(* IEC 61131-3 sources: programs/VI-54/VI-54_20171205/VI-54_20171205/Stations/PLC_VI54/VI-54_171014/Class/SdiasManager (part 2) *)

              // additional info which may be needed by the module
              tempCmd.aPara[2] := ud_BusTime_ns$DINT;
              tempCmd.aPara[3] := to_dint(ManagerInfoBlock.ModuleInfos[ActInitAccessIndex].FPGAVersion);

              // check if device ID is ok
              if pModuleInfo^.pThis^.NewInst(pPara:=#tempCmd, pResult:=#_result) = READY then

                // update default accesses if available
                if ManagerInfoBlock.ModuleInfos[ActInitAccessIndex].ReadAccess.usLength then
                  pModuleInfo^.pDefaultAccesses^.ReadAccess.hiOffset := ManagerInfoBlock.ModuleInfos[ActInitAccessIndex].ReadAccess.hiOffset;
                  pModuleInfo^.pDefaultAccesses^.ReadAccess.usLength := ManagerInfoBlock.ModuleInfos[ActInitAccessIndex].ReadAccess.usLength;
                end_if;

                if ManagerInfoBlock.ModuleInfos[ActInitAccessIndex].WriteAccess.usLength then
                  pModuleInfo^.pDefaultAccesses^.WriteAccess.hiOffset := ManagerInfoBlock.ModuleInfos[ActInitAccessIndex].WriteAccess.hiOffset;
                  pModuleInfo^.pDefaultAccesses^.WriteAccess.usLength := ManagerInfoBlock.ModuleInfos[ActInitAccessIndex].WriteAccess.usLength;
                end_if;

                tempCmd.uiCmd := SDIAS_CMD_INIT_ACCESSES;
                RetcodeIPR := pModuleInfo^.pThis^.NewInst(pPara:=#tempCmd, pResult:=#_result);
                if RetcodeIPR = BUSY then
                  // if any module needs more runs => continue here next time
                  b_ModulInitFinished := FALSE;
                  exit;
                elsif RetcodeIPR = ERROR then
                  LogValue("(SdiasManager::CyWork) Failed to add accesses on SDIAS Place 0x{0}", ActInitAccessIndex);
                end_if;
              end_if;
            end_if;
            pModuleInfo += sizeof(t_ModuleObjectInfo);
            ActInitAccessIndex += 1;
          end_while;
        end_if;

        // if we got all accesse => go on
        if b_ModulInitFinished then
          // only if there are entries
          if ManagerInfoBlock.MappingInfo.MappingInfoNo then
            // if the post init is over and the DOs are not created yet => create them in Rt-SSW
            if b_PostInitFinished then
              InitSSW := _StartRtIsoDOCreation;
            else
              CreateAndModifyIsoDOs();

              InitSSW := _CheckInfoBlock;
            end_if;
          else
            LogError("(SdiasManager::CyWork) No Mapping Info in Info Block of SDIAS Manager found! Unable to continue Initialisation!");
            ErrorInitStep := InitSSW;
            InitSSW := _PrepareError;
            ClassState := _ComponentNotExists;
          end_if;
        end_if;

//**********************************************************************************************************************************************************
      _StartRtIsoDOCreation:
        // create and modify the iso DOs in realtime priority
        RtSSW := _CreateAndModifyDOs;
        InitSSW := _Wait4RtIsoDOCreation;

//**********************************************************************************************************************************************************
      _Wait4RtIsoDOCreation:
        // wait for the DOs to be ready
        if RtSSW = _Wait4DOs then
          InitSSW := _CheckInfoBlock;
        end_if;

//**********************************************************************************************************************************************************
      _CheckInfoBlock:

        // only if there are entries
        if ManagerInfoBlock.MappingInfo.MappingInfoNo then
          if ISOWriteDO.pData & ISOReadDO.pData then

            // on VIs the info is copied into the payload. on local SDIAS we get the info directly from the OS
            if ConnectionType = SDIAS_CON_VIA_VARAN_uC then
              pTaskHelp := TaskInfoDO.pData$^t_TaskInfoReadData;
              WriteTaskInfo.pReadData := #pTaskHelp^.WriteTaskInfo;
              ReadTaskInfo.pReadData  := #pTaskHelp^.ReadTaskInfo;
            else
              WriteTaskInfo.pReadData := #WrTaskInfo;
              ReadTaskInfo.pReadData  := #RdTaskInfo;
            end_if;

            // tell the modules their DeviceID, Serialnumber and check if it's the correct object at this place. if so, give them the access pointers
            pModuleInfo := #ModuleObjInfo[0];
            for i := 0 to MaxPlace do

              // if we have an object with this place
              if pModuleInfo^.pThis then
                // and the µC detected a module at this place
                if IsDeviceBitSet(pDeviceBitMap:=#HardwareConfig.DeviceBitmap[0], Place:=i) then

                  if ManagerInfoBlock.ModuleInfos[i].ModuleID = 16#FFFF then
                    pModuleInfo^.pInitState^ := _SPIError;
                  else
                    // get the init state of the LED of this object
                    TempLEDState := pModuleInfo^.pThis^.LEDControl$USINT;

                    // save the state in the local LED Image

                    // get byte position ouf of place (place 0-3 in byte 0, 4-7 in byte 1,...)
                    ByteNr := i$USINT SHR 2;
                    PosInByte := (i$USINT AND 2#11) SHL 1;
                    AppliLEDStates[ByteNr] := (AppliLEDStates[ByteNr] AND NOT(2#11 SHL PosInByte)) OR (TempLEDState SHL PosInByte);

                    // new device info with length parameter to ensure compatibility
                    tempCmd.uiCmd := SDIAS_CMD_DEVICE_INFO2;
                    tempCmd.aPara[0] := sizeof(HDINT); // length of following parameters

                    // hardware version: for 1.10 (printed on the module) we have to transform 16#01 major and 16#0100 minor (drop high nibbles of minor) to 16#00000110
                    tempCmd.aPara[1] := to_dint((ManagerInfoBlock.ModuleInfos[i].HWVersion SHL 8)            OR
                                        ((ManagerInfoBlock.ModuleInfos[i].HWVersionMidLow  SHR 4) AND 16#F0) OR
                                        ((ManagerInfoBlock.ModuleInfos[i].HWVersionMidLow       ) AND 16#0F));

                    // don't check the return code since this command may not be supported
                    pModuleInfo^.pThis^.NewInst(pPara:=#tempCmd, pResult:=#_result);

                    // send the device info to the module
                    tempCmd.uiCmd := SDIAS_CMD_DEVICE_INFO;
                    tempCmd.aPara[0] := to_dint(ManagerInfoBlock.ModuleInfos[i].ModuleID);
                    tempCmd.aPara[1] := (#ManagerInfoBlock.ModuleInfos[i].SerialNo[0])$DINT;

                    // additional info which may be needed by the module
                    tempCmd.aPara[2] := ud_BusTime_ns$DINT;
                    tempCmd.aPara[3] := to_dint(ManagerInfoBlock.ModuleInfos[i].FPGAVersion);

                    // check if device ID is ok
                    if pModuleInfo^.pThis^.NewInst(pPara:=#tempCmd, pResult:=#_result) = READY then

                      // the module id matches, now check the accesses

                      // update default accesses if available
                      if ManagerInfoBlock.ModuleInfos[i].ReadAccess.usLength then
                        pModuleInfo^.pDefaultAccesses^.ReadAccess.hiOffset := ManagerInfoBlock.ModuleInfos[i].ReadAccess.hiOffset;
                        pModuleInfo^.pDefaultAccesses^.ReadAccess.usLength := ManagerInfoBlock.ModuleInfos[i].ReadAccess.usLength;

                        // store the pointers to the correct payload data for later usage in the SDIAS Client class
                        pModuleInfo^.pDefaultAccesses^.ReadAccess.pControlByte$^void  := ISOWriteDO.pData + ManagerInfoBlock.ModuleInfos[i].ReadDODataWrOffset - ISOWriteDO.Offset;
                        pModuleInfo^.pDefaultAccesses^.ReadAccess.pStateByte$^void    := ISOReadDO.pData  + ManagerInfoBlock.ModuleInfos[i].ReadDODataRdOffset - ISOReadDO.Offset;
                        pModuleInfo^.pDefaultAccesses^.ReadAccess.pData               := ISOReadDO.pData  + ManagerInfoBlock.ModuleInfos[i].ReadDODataRdOffset - ISOReadDO.Offset + sizeof(t_SDIAS_StateByte);
                      end_if;

                      if ManagerInfoBlock.ModuleInfos[i].WriteAccess.usLength then
                        pModuleInfo^.pDefaultAccesses^.WriteAccess.hiOffset := ManagerInfoBlock.ModuleInfos[i].WriteAccess.hiOffset;
                        pModuleInfo^.pDefaultAccesses^.WriteAccess.usLength := ManagerInfoBlock.ModuleInfos[i].WriteAccess.usLength;

                        // store the pointers to the correct payload data for later usage in the SDIAS Client class
                        pModuleInfo^.pDefaultAccesses^.WriteAccess.pControlByte$^void  := ISOWriteDO.pData + ManagerInfoBlock.ModuleInfos[i].WriteDODataWrOffset - ISOWriteDO.Offset;
                        pModuleInfo^.pDefaultAccesses^.WriteAccess.pStateByte$^void    := ISOReadDO.pData + ManagerInfoBlock.ModuleInfos[i].WriteDODataRdOffset - ISOReadDO.Offset;
                        pModuleInfo^.pDefaultAccesses^.WriteAccess.pData               := ISOWriteDO.pData + ManagerInfoBlock.ModuleInfos[i].WriteDODataWrOffset - ISOWriteDO.Offset + sizeof(t_SDIAS_ControlByte);
                      end_if;
                    else
                      // wrong device ID
                      if pModuleInfo^.Required then
                        // first stop blocking the init, otherwise the init freezes when we have a required error
                        if b_PostInitFinished = FALSE then
                          SendPostInitFinished(DisableThisObject:=TRUE);
                        end_if;

                        LogValue("(SdiasManager::CyWork) Wrong device ID at SDIAS Place 0x{0}", i);

                        SetRequiredError(pTargetThis:=pModuleInfo^.pThis, Place:=i);
                      else
                        pModuleInfo^.pInitState^ := _WrongHardware;
                      end_if;
                    end_if;
                  end_if;
                else
                  // module is not in the device bitmap, but we got an object
                  if pModuleInfo^.Required then
                    // first stop blocking the init, otherwise the init freezes when we have a required error
                    if b_PostInitFinished = FALSE then
                      SendPostInitFinished(DisableThisObject:=TRUE);
                    end_if;

                    SetRequiredError(pTargetThis:=pModuleInfo^.pThis, Place:=i);
                  else
                    pModuleInfo^.pInitState^ := _NoHardware;
                  end_if;
                end_if;
              end_if;

              pModuleInfo += sizeof(t_ModuleObjectInfo);
            end_for;
          end_if;

          if ConnectionType = SDIAS_CON_VIA_VARAN_uC then
            InitSSW := _PrepareResetIsoRdPayload;
          else
            // we don't have to reset the payload => done by OS
            udCurCheckedMod := 0;
            InitSSW := _CheckModule_Valid;
          end_if;

        else
          LogError("(SdiasManager::CyWork) No Mapping Info in Info Block of SDIAS Manager found! Unable to continue Initialisation!");
          ErrorInitStep := InitSSW;
          InitSSW := _PrepareError;
          ClassState := _ComponentNotExists;
        end_if;

//**********************************************************************************************************************************************************
      _PrepareResetIsoRdPayload:
        // prepare resetting the read payload (toggle bits)
        AccessProgress := 0;
        // reset the write buffer
        _memset(dest:=ASYWriteDO.pData, usByte:=0, cntr:=128);
        NewDataSize := ISOReadDO.Length;
        if NewDataSize > 128 then
          NewDataSize := 128;
        end_if;

        if ChangeAsyWr(Offset:=ISOReadDO.Offset,
                       Length:=NewDataSize$USINT,
                       RunState:=_BUS_IF_RUN_STATE_CONT_RUN,
                       UsageType:=_UsedBySSW) then

          InitSSW := _ResetIsoRdPayload;
        end_if;

//**********************************************************************************************************************************************************
      _ResetIsoRdPayload:
        AccessProgress += NewDataSize;

        if AccessProgress < ISOReadDO.Length then
          if (ISOReadDO.Length - AccessProgress) > 128 then
            // we need more than 128 bytes => write the next 128
            TempNewDataSize := 128;
          else
            // we need to write the rest (last package)
            TempNewDataSize := (ISOReadDO.Length - AccessProgress);
          end_if;

          if ChangeAsyWr(Offset:=ISOReadDO.Offset + AccessProgress,
                         Length:=TempNewDataSize$USINT,
                         RunState:=_BUS_IF_RUN_STATE_CONT_RUN,
                         UsageType:=_UsedBySSW) then
              NewDataSize := TempNewDataSize;
          else
            NewDataSize := 0;
          end_if;
        else
          // we got the complete info block now => stop the DO
          if ChangeAsyWr(Offset:=0,
                         Length:=0,
                         RunState:=_BUS_IF_RUN_STATE_NO_RUN,
                         UsageType:=_UsedBySSW) then

            InitSSW := _PrepareResetIsoWrPayload;
          else
            NewDataSize := 0;
          end_if;
        end_if;

//**********************************************************************************************************************************************************
      _PrepareResetIsoWrPayload:
        // prepare resetting the read payload (toggle bits)
        AccessProgress := 0;
        // reset the write buffer
        _memset(dest:=ASYWriteDO.pData, usByte:=0, cntr:=128);
        NewDataSize := ISOWriteDO.Length;
        if NewDataSize > 128 then
          NewDataSize := 128;
        end_if;

        if ChangeAsyWr(Offset:=ISOWriteDO.Offset,
                       Length:=NewDataSize$USINT,
                       RunState:=_BUS_IF_RUN_STATE_CONT_RUN,
                       UsageType:=_UsedBySSW) then

          InitSSW := _ResetIsoWrPayload;
        end_if;

//**********************************************************************************************************************************************************
      _ResetIsoWrPayload:
        AccessProgress += NewDataSize;

        if AccessProgress < ISOWriteDO.Length then
          if (ISOWriteDO.Length - AccessProgress) > 128 then
            // we need more than 128 bytes => write the next 128
            TempNewDataSize := 128;
          else
            // we need to write the rest (last package)
            TempNewDataSize := (ISOWriteDO.Length - AccessProgress);
          end_if;

          if ChangeAsyWr(Offset:=ISOWriteDO.Offset + AccessProgress,
                         Length:=TempNewDataSize$USINT,
                         RunState:=_BUS_IF_RUN_STATE_CONT_RUN,
                         UsageType:=_UsedBySSW) then
              NewDataSize := TempNewDataSize;
          else
            NewDataSize := 0;
          end_if;
        else
          // we got the complete info block now => stop the DO
          if ChangeAsyWr(Offset:=0,
                         Length:=0,
                         RunState:=_BUS_IF_RUN_STATE_NO_RUN,
                         UsageType:=_UsedBySSW) then

            udCurCheckedMod := 0;
            InitSSW := _CheckModule_Valid;
          else
            NewDataSize := 0;
          end_if;
        end_if;

//**********************************************************************************************************************************************************
      _CheckModule_Valid:
        // tell the modules their DeviceID, Serialnumber and check if it's the correct object at this place. if so, give them the access pointers
        pModuleInfo := #ModuleObjInfo[udCurCheckedMod];

        // if we have an object with this place
        if pModuleInfo^.pThis then
          // and the µC detected a module at this place
          if IsDeviceBitSet(pDeviceBitMap:=#HardwareConfig.DeviceBitmap[0], Place:=udCurCheckedMod) then

            if ManagerInfoBlock.ModuleInfos[udCurCheckedMod].ModuleID = 16#FFFF then
              // SPI Error
              if pModuleInfo^.Required then
                // first stop blocking the init, otherwise the init freezes when we have a required error
                if b_PostInitFinished = FALSE then
                  SendPostInitFinished(DisableThisObject:=TRUE);
                end_if;

                LogValue("(SdiasManager::CyWork) Wrong device ID at SDIAS Place 0x{0}", udCurCheckedMod);

                SetRequiredError(pTargetThis:=pModuleInfo^.pThis, Place:=udCurCheckedMod);
              else
                pModuleInfo^.pInitState^ := _SPIError;
                InitSSW := _CheckNextModule;
              end_if;
            else
              // get the init state of the LED of this object
              TempLEDState := pModuleInfo^.pThis^.LEDControl$USINT;

              // save the state in the local LED Image

              // get byte position ouf of place (place 0-3 in byte 0, 4-7 in byte 1,...)
              ByteNr := udCurCheckedMod$USINT SHR 2;
              PosInByte := (udCurCheckedMod$USINT AND 2#11) SHL 1;
              AppliLEDStates[ByteNr] := (AppliLEDStates[ByteNr] AND NOT(2#11 SHL PosInByte)) OR (TempLEDState SHL PosInByte);

              // new device info with length parameter to ensure compatibility
              tempCmd.uiCmd := SDIAS_CMD_DEVICE_INFO2;
              tempCmd.aPara[0] := sizeof(HDINT); // length of following parameters

              // hardware version: for 1.10 (printed on the module) we have to transform 16#01 major and 16#0100 minor (drop high nibbles of minor) to 16#00000110
              tempCmd.aPara[1] := to_dint((ManagerInfoBlock.ModuleInfos[udCurCheckedMod].HWVersion SHL 8)            OR
                                  ((ManagerInfoBlock.ModuleInfos[udCurCheckedMod].HWVersionMidLow  SHR 4) AND 16#F0) OR
                                  ((ManagerInfoBlock.ModuleInfos[udCurCheckedMod].HWVersionMidLow       ) AND 16#0F));

              // don't check the return code since this command may not be supported
              pModuleInfo^.pThis^.NewInst(pPara:=#tempCmd, pResult:=#_result);

              // send the device info to the module
              tempCmd.uiCmd := SDIAS_CMD_DEVICE_INFO;
              tempCmd.aPara[0] := to_dint(ManagerInfoBlock.ModuleInfos[udCurCheckedMod].ModuleID);
              tempCmd.aPara[1] := (#ManagerInfoBlock.ModuleInfos[udCurCheckedMod].SerialNo[0])$DINT;

              // additional info which may be needed by the module
              tempCmd.aPara[2] := ud_BusTime_ns$DINT;
              tempCmd.aPara[3] := to_dint(ManagerInfoBlock.ModuleInfos[udCurCheckedMod].FPGAVersion);

              // check if device ID is ok
              if pModuleInfo^.pThis^.NewInst(pPara:=#tempCmd, pResult:=#_result) = READY then

                // the module id matches, continue with access
                pCurCheckModAccPtr := pModuleInfo^.pFirstAccess;
                InitSSW := _SetModAccess;

              else
                // wrong device ID
                if pModuleInfo^.Required then
                  // first stop blocking the init, otherwise the init freezes when we have a required error
                  if b_PostInitFinished = FALSE then
                    SendPostInitFinished(DisableThisObject:=TRUE);
                  end_if;

                  LogValue("(SdiasManager::CyWork) Wrong device ID at SDIAS Place 0x{0}", udCurCheckedMod);

                  SetRequiredError(pTargetThis:=pModuleInfo^.pThis, Place:=udCurCheckedMod);
                else
                  pModuleInfo^.pInitState^ := _WrongHardware;
                  InitSSW := _CheckNextModule;
                end_if;
              end_if;
            end_if;
          else
            // module is not in the device bitmap, but we got an object
            if pModuleInfo^.Required then
              // first stop blocking the init, otherwise the init freezes when we have a required error
              if b_PostInitFinished = FALSE then
                SendPostInitFinished(DisableThisObject:=TRUE);
              end_if;

              SetRequiredError(pTargetThis:=pModuleInfo^.pThis, Place:=udCurCheckedMod);
            else
              pModuleInfo^.pInitState^ := _NoHardware;
              InitSSW := _CheckNextModule;
            end_if;
          end_if;
        else
          InitSSW := _CheckNextModule;
        end_if;

//**********************************************************************************************************************************************************
      _SetModAccess:
        pModuleInfo := #ModuleObjInfo[udCurCheckedMod];
        if pCurCheckModAccPtr = NIL then
          // no special accesses => call connect event and proceed with next module
          pModuleInfo^.pThis^.ConnectEvent();
          InitSSW := _CheckNextModule;
        elsif (pCurCheckModAccPtr^.eAccessType = _Read) | (pCurCheckModAccPtr^.eAccessType = _ReadDynamic) then

          pWaitAccess := pCurCheckModAccPtr^.pWaitForAccess;
          if pWaitAccess <> NIL then
            if (pWaitAccess^.eAccessType <> pCurCheckModAccPtr^.eAccessType) then
              pWaitAccess := NIL;
            end_if;
          end_if;

          if(pWaitAccess <> NIL) then
            // address of state byte
            iWaitOffset := ISOReadDO.Offset + (pWaitAccess^.ppStateByte^$HDINT - ISOReadDO.pData$HDINT)$UINT; //pWaitAccess^.hiDOOffsetInDPRAM;
          else
            iWaitOffset := SDIAS_INVALID_VOLATILE_WAIT_HANDLE;
          end_if;

          // Create access by new funtion
          iRetCode := DOL_Handling_Add_DO_TO_List(bIsWriteAcc0:= 0,
                                                  iModAddr0:= pCurCheckModAccPtr^.hiOffset + (udCurCheckedMod shl 10),
                                                  iDataLen0:= pCurCheckModAccPtr^.uiLength,
                                                  bCtrlAcc0:= pCurCheckModAccPtr^.bCtrlAcc0,
                                                  iWaitDOOffset0:= iWaitOffset,
                                                  bIsDynamic0 := (pCurCheckModAccPtr^.eAccessType = _ReadDynamic),
                                                  pActAccess0 := pCurCheckModAccPtr);

          if iRetCode = 0 then

            // store the pointers to the correct payload data for later usage in the SDIAS Client class
            if pCurCheckModAccPtr^.ppControlByte then
              pCurCheckModAccPtr^.ppControlByte^$^void := ISOWriteDO.pData + gcWrite_DOL_Desc.iOffFirstData + gcMapping_Informations[IsoWrPayload].StartAddress - ISOWriteDO.Offset;
              if pCurCheckModAccPtr^.eAccessType = _ReadDynamic then
                pControlStruct := pCurCheckModAccPtr^.ppControlByte^$^t_SDIAS_ControlStructDynamic;
                pControlStruct^.ControlByte.EnableFlexRead := TRUE;
                pControlStruct^.hiOffset := pCurCheckModAccPtr^.hiOffset + (udCurCheckedMod shl 10);
                pControlStruct^.usLength := pCurCheckModAccPtr^.uiLength$USINT;
              end_if;
            end_if;
            if pCurCheckModAccPtr^.ppStateByte then
              pCurCheckModAccPtr^.ppStateByte^$^void := ISOReadDO.pData + gcRead_DOL_Desc.iOffFirstData + gcMapping_Informations[IsoRdPayload].StartAddress - ISOReadDO.Offset;
            end_if;
            if pCurCheckModAccPtr^.ppData then
              pCurCheckModAccPtr^.ppData^$^void := ISOReadDO.pData + gcRead_DOL_Desc.iOffFirstData + sizeof(t_SDIAS_StateByte) + gcMapping_Informations[IsoRdPayload].StartAddress - ISOReadDO.Offset;;
            end_if;

            InitSSW := _WriteModAccess;
          else
            ErrorInitStep := InitSSW;
            InitSSW := _PrepareError;
            ClassState := _DOCmdInvalid;
          end_if;

        elsif (pCurCheckModAccPtr^.eAccessType = _Write) | (pCurCheckModAccPtr^.eAccessType = _WriteDynamic) then

          pWaitAccess := pCurCheckModAccPtr^.pWaitForAccess;
          if pWaitAccess <> NIL then
            if (pWaitAccess^.eAccessType <> pCurCheckModAccPtr^.eAccessType) then
              pWaitAccess := NIL;
            end_if;
          end_if;

          if(pWaitAccess <> NIL) then
            // address of state byte
            iWaitOffset := ISOReadDO.Offset + (pWaitAccess^.ppStateByte^$HDINT - ISOReadDO.pData$HDINT)$UINT; //pWaitAccess^.hiDOOffsetInDPRAM;
          else
            iWaitOffset := SDIAS_INVALID_VOLATILE_WAIT_HANDLE;
          end_if;

          // Create access by new funtion
          iRetCode := DOL_Handling_Add_DO_TO_List(bIsWriteAcc0:= 1,
                                                  iModAddr0:= pCurCheckModAccPtr^.hiOffset + (udCurCheckedMod shl 10),
                                                  iDataLen0:= pCurCheckModAccPtr^.uiLength,
                                                  bCtrlAcc0:= pCurCheckModAccPtr^.bCtrlAcc0,
                                                  iWaitDOOffset0:= iWaitOffset,
                                                  bIsDynamic0 := (pCurCheckModAccPtr^.eAccessType = _WriteDynamic),
                                                  pActAccess0 := pCurCheckModAccPtr);

          if iRetCode = 0 then
            // store the pointers to the correct payload data for later usage in the SDIAS Client class
            if pCurCheckModAccPtr^.ppControlByte then
              pCurCheckModAccPtr^.ppControlByte^$^void := ISOWriteDO.pData + gcWrite_DOL_Desc.iOffFirstData + gcMapping_Informations[IsoWrPayload].StartAddress - ISOWriteDO.Offset;
              if pCurCheckModAccPtr^.eAccessType = _WriteDynamic then
                pControlStruct := pCurCheckModAccPtr^.ppControlByte^$^t_SDIAS_ControlStructDynamic;
                pControlStruct^.ControlByte.EnableFlexWrite := TRUE;
                pControlStruct^.hiOffset := pCurCheckModAccPtr^.hiOffset + (udCurCheckedMod shl 10);
                pControlStruct^.usLength := pCurCheckModAccPtr^.uiLength$USINT;
              end_if;
            end_if;
            if pCurCheckModAccPtr^.ppStateByte then
              pCurCheckModAccPtr^.ppStateByte^$^void := ISOReadDO.pData + gcRead_DOL_Desc.iOffFirstData + gcMapping_Informations[IsoRdPayload].StartAddress - ISOReadDO.Offset;
            end_if;
            if pCurCheckModAccPtr^.ppData then
              // the data start after the header. at dynamic objects we have more header in write payload => data start after the structure
              if pCurCheckModAccPtr^.eAccessType = _WriteDynamic then
                pCurCheckModAccPtr^.ppData^$^void := ISOWriteDO.pData + gcWrite_DOL_Desc.iOffFirstData + sizeof(t_SDIAS_ControlStructDynamic) + gcMapping_Informations[IsoWrPayload].StartAddress - ISOWriteDO.Offset;
              else
                pCurCheckModAccPtr^.ppData^$^void := ISOWriteDO.pData + gcWrite_DOL_Desc.iOffFirstData + sizeof(t_SDIAS_ControlByte) + gcMapping_Informations[IsoWrPayload].StartAddress - ISOWriteDO.Offset;
              end_if;
            end_if;

            InitSSW := _WriteModAccess;
          else
            ErrorInitStep := InitSSW;
            InitSSW := _PrepareError;
            ClassState := _DOCmdInvalid;
          end_if;
        end_if;

//**********************************************************************************************************************************************************
      _WriteModAccess:

          if ConnectionType = SDIAS_CON_VIA_VARAN_uC then
            ASYWriteDO.pData^$t_SDIAS_DOListEntryX2 := cModulAccessCmds;

            // Write data to manager dpram
            if ChangeAsyWr(Offset   := uiWriteCmdAddr,
                           Length   := sizeof(cModulAccessCmds),
                           RunState := _BUS_IF_RUN_STATE_SINGLE_RUN,
                           UsageType:= _UsedBySSW) then

              InitSSW := _SetNextModAccess;
            end_if;
          else
            // OS already did this for us
            InitSSW := _SetNextModAccess;
          end_if;

//**********************************************************************************************************************************************************
      _SetNextModAccess:

        AsyWriteUsage  := _NotUsed;

        pModuleInfo := #ModuleObjInfo[udCurCheckedMod];
        // Reached last access - trigger connect event
        if(pCurCheckModAccPtr^.pNext = NIL) then
          // call the connect event now (pointers are set now to enable the accesses)
          pModuleInfo^.pThis^.ConnectEvent();
          InitSSW := _CheckNextModule;
        else
          pCurCheckModAccPtr := pCurCheckModAccPtr^.pNext;
          InitSSW := _SetModAccess;
        end_if;

//**********************************************************************************************************************************************************
      _CheckNextModule:

        // Switch to next module
        udCurCheckedMod += 1;

        if(udCurCheckedMod <= MaxPlace) then
          InitSSW := _CheckModule_Valid;
        else
          if ConnectionType = SDIAS_CON_VIA_VARAN_uC then
            InitSSW := _WriteDOL_Offsets;
          else
            // we don't have to reset the payload => done by OS
            if MaxPlace <> SDIAS_PLACE_NO_MODULE_ADDED_SO_FAR then
              InitSSW := _SetStartConfigIsoRd;
            else
              LogError("(SdiasManager::CyWork) No SDIAS Client objects projected/connected to the SDIAS Manager! Unable to continue with Initialisation!");
              ErrorInitStep := InitSSW;
              InitSSW := _PrepareError;
              ClassState := _NoHardware;
            end_if;
          end_if;
        end_if;

//**********************************************************************************************************************************************************
      _WriteDOL_Offsets:

        // Create list informations
        // Read list offsets
        iDataOffsets[0] := gcRead_DOL_Desc.iOffEndCmd;
        iDataOffsets[1] := gcRead_DOL_Desc.iOffLastData;

        // Write list offsets
        iDataOffsets[2] := gcWrite_DOL_Desc.iOffEndCmd;
        iDataOffsets[3] := gcWrite_DOL_Desc.iOffLastData;

        bReceivedNewEndRsp := FALSE;
#ifdef HWK_SHOW_PRAGMA_MESSAGES
#pragma message("RamAnd 23.11.2013 19:17 \ ein neues Ende muss nur geschrieben werden, wenn Spezialzugriffe angelegt wurden")
#endif
        if(AddSDOReq(pCmdSvr:= (#ClassState.pMeth)$^SvrChCmd,
                     Command:= SDIAS_SDO_CMD_SET_NEW_END,
                     Place:= SDIAS_MANAGER_PLACE,
                     CmdLength:= 4* sizeof(UDINT),
                     pReqBuf:= #iDataOffsets[0]$USINT) = READY$DINT) then

           InitSSW := _WaitReq_DOL_Offsets;
        end_if;

//**********************************************************************************************************************************************************
      _WaitReq_DOL_Offsets:
        // Wait until receiving request
        if bReceivedNewEndRsp = TRUE then
          bReceivedNewEndRsp := FALSE;

          InitSSW := _GetEventIDs;
        end_if;

//**********************************************************************************************************************************************************
      _GetEventIDs:
        if MaxPlace <> SDIAS_PLACE_NO_MODULE_ADDED_SO_FAR then
            // we also start a read access here, so we got the data in the next step
          if ChangeAsyRd(Offset:=SDIAS_OFFSET_TASK_EVENT_IDS,
                         Length:=sizeof(t_TaskEventIDs),
                         RunState:=_BUS_IF_RUN_STATE_SINGLE_RUN,
                         UsageType:=_UsedBySSW) then

            udCurCheckedMod := 0;
            InitSSW := _SetStartConfigIsoRd;
          end_if;
        else
          LogError("(SdiasManager::CyWork) No SDIAS Client objects projected/connected to the SDIAS Manager! Unable to continue with Initialisation!");
          ErrorInitStep := InitSSW;
          InitSSW := _PrepareError;
          ClassState := _NoHardware;
        end_if;

//**********************************************************************************************************************************************************
      _SetStartConfigIsoRd:
        if ConnectionType = SDIAS_CON_VIA_VARAN_uC then
          TaskEventIDs := ASYReadDO.pData^$t_TaskEventIDs;
        else
          for i := 0 to 7 do
            if SDIAS_iGetNodePropertyIndex(hNodeHandle    := udNodeHandle
                                    , udIndex             := i
                                    , udPropertyId        := SDM_PROP_TASK_START_EVENT_ID,
                                    , pudPropertyValue    := (#TaskEventIDs[i])$^UDINT
                                    ) <> SDIAS_OK then
              LogValue("(SdiasManager::CyWork) Failed to get task event ID 0x{0} via OS interface!", i);
              ErrorInitStep := InitSSW;
              InitSSW := _PrepareError;
              ClassState := _ManagerError;
              return;
            end_if;
          end_for;
        end_if;

        AsyReadUsage  := _NotUsed;

        // search for the sync out 0 event id
        b_FoundIt := FALSE;
        for i := 0 to 7 do
          if ConnectionType = SDIAS_CON_VIA_VARAN_uC then
            if TaskEventIDs[i] = SDIAS_EVENT_MASK_ID_SYNC_OUT0 then
              b_FoundIt := TRUE;
              exit;
            end_if;
          else
            if TaskEventIDs[i] = SDIAS_EVENT_MASK_ID_SYNC_OUT2 then
              b_FoundIt := TRUE;
              exit;
            end_if;
          end_if;
        end_for;

        // if we found it, use it for the task start config 0 (which is used by the iso read task)
        if b_FoundIt then
          TaskStartConfig.EventSelection := 1 SHL i$USINT;

          // iso read starts 0µs after the sync
          TaskStartConfig.StartDelay_us  := 0;

          if ConnectionType = SDIAS_CON_VIA_VARAN_uC then
            ASYWriteDO.pData^$t_TaskStartConfig := TaskStartConfig;
            if ChangeAsyWr(Offset:=SDIAS_OFFSET_TASK_START_CFG_0,
                           Length:=sizeof(t_TaskStartConfig),
                           RunState:=_BUS_IF_RUN_STATE_SINGLE_RUN,
                           UsageType:=_UsedBySSW) then

             InitSSW := _SelectTaskStartConfigIsoRd;
            end_if;
          else
            aProperties[0].udPropertyId     := SDM_PROP_TASK_START_CONFIG_WAIT_EVENTS;
            aProperties[0].udPropertyValue  := TaskStartConfig.EventSelection;

            aProperties[1].udPropertyId     := SDM_PROP_TASK_START_CONFIG_DELAY;
            aProperties[1].udPropertyValue  := TaskStartConfig.StartDelay_us;

            if SDIAS_iSetNodePropertiesIndex(hNodeHandle      := udNodeHandle
                                           , udIndex               := 0
                                           , udPropertyCount       := 2
                                           , psPropertyValuePairs  := #aProperties[0]
                                           ) = SDIAS_OK then
              InitSSW := _SelectTaskStartConfigIsoRd;
            else
              LogError("(SdiasManager::CyWork) Failed to set the iso read start config via OS interface!");
              ErrorInitStep := InitSSW;
              InitSSW := _PrepareError;
              ClassState := _ManagerError;
            end_if;
          end_if;
        else
          LogError("(SdiasManager::CyWork) Couldn't find event mask of sync out 0! Unable to continue with Initialisation!");
          ClassState := _ComponentNotExists;
          ErrorInitStep := InitSSW;
          InitSSW := _PrepareError;
        end_if;

//**********************************************************************************************************************************************************
      _SelectTaskStartConfigIsoRd:
        // search for the iso read entry in the info block
        b_FoundIt := FALSE;
        for i := 0 to ManagerInfoBlock.MappingInfo.MappingInfoNo-1 do
          if ManagerInfoBlock.MappingInfo.aMappingInfos[i].MappingID = IsoRdList then
            b_FoundIt := TRUE;
            exit;
          end_if;
        end_for;

        // if we found it, use the offset in the task configuration
        if b_FoundIt then
          // set the task duration limit
          TaskConfig.TaskDurationTimeout_us := (ud_BusTime_ns / 1000)$UINT;
#ifdef HWK_SHOW_PRAGMA_MESSAGES
#pragma message("RamAnd 21.10.2013 17:46 \ Timeoutzeit überdenken. hier kann normalerweise kein ganzer Buszyklus verwendet werden (IsoStartpoint miteinbeziehen)")
#endif

          // start address of iso read list
          TaskConfig.Config := ManagerInfoBlock.MappingInfo.aMappingInfos[i].StartAddress;

          // now select the start configuration 0 (should already be selected, just check it)
          if TaskConfig.Config AND 2#1111 then
            // in this case the start address of the list is not 16 byte aligned
            LogError("(SdiasManager::CyWork) The start address of the isochronous read DO List is not 16 byte aligned! Unable to continue with Initialisation!");
            ClassState := _MemoryFault;
            ErrorInitStep := InitSSW;
            InitSSW := _PrepareError;
            return;
          end_if;

          // we want to use the start configuration => enable it later in realtime
          TaskConfig.Config.SynchronizedStartEnable := FALSE;

          if ConnectionType = SDIAS_CON_VIA_VARAN_uC then
            ASYWriteDO.pData^$t_TaskConfig := TaskConfig;

            if ChangeAsyWr(Offset:=SDIAS_OFFSET_TASK_CONFIG_1,
                           Length:=sizeof(t_TaskConfig),
                           RunState:=_BUS_IF_RUN_STATE_SINGLE_RUN,
                           UsageType:=_UsedBySSW) then

              InitSSW := _SelectTaskStartConfigIsoWr;
            end_if;
          else
            aProperties[0].udPropertyId     := SDM_PROP_TASK_CONTROL_DURATION_TIMEOUT;
            aProperties[0].udPropertyValue  := TaskConfig.TaskDurationTimeout_us;

            aProperties[1].udPropertyId     := SDM_PROP_TASK_CONTROL_CONFIGURATION;
            aProperties[1].udPropertyValue  := TaskConfig.Config;

            if SDIAS_iSetNodePropertiesIndex(hNodeHandle      := udNodeHandle
                                      , udIndex               := 1
                                      , udPropertyCount       := 2
                                      , psPropertyValuePairs  := #aProperties[0]
                                      ) = SDIAS_OK then
              InitSSW := _SelectTaskStartConfigIsoWr;
            else
              LogError("(SdiasManager::CyWork) Failed to set the iso read start config via OS interface!");
              ErrorInitStep := InitSSW;
              InitSSW := _PrepareError;
              ClassState := _ManagerError;
            end_if;

          end_if;
        else
          LogError("(SdiasManager::CyWork) Couldn't find iso read entry in info block! Unable to continue with Initialisation!");
          ClassState := _ComponentNotExists;
          ErrorInitStep := InitSSW;
          InitSSW := _PrepareError;
        end_if;

//**********************************************************************************************************************************************************
      _SelectTaskStartConfigIsoWr:
        // search for the iso write entry in the info block
        b_FoundIt := FALSE;
        for i := 0 to ManagerInfoBlock.MappingInfo.MappingInfoNo-1 do
          if ManagerInfoBlock.MappingInfo.aMappingInfos[i].MappingID = IsoWrList then
            b_FoundIt := TRUE;
            exit;
          end_if;
        end_for;

        // if we found it, use the offset in the task configuration
        if b_FoundIt then
          // set the task duration limit
          TaskConfig.TaskDurationTimeout_us := (ud_BusTime_ns / 1000)$UINT;

          // start address of iso write list
          TaskConfig.Config := ManagerInfoBlock.MappingInfo.aMappingInfos[i].StartAddress;

          if ConnectionType = SDIAS_CON_VIA_VARAN_uC then
            ASYWriteDO.pData^$t_TaskConfig := TaskConfig;

            if ChangeAsyWr(Offset:=SDIAS_OFFSET_TASK_CONFIG_2,
                           Length:=sizeof(t_TaskConfig),
                           RunState:=_BUS_IF_RUN_STATE_SINGLE_RUN,
                           UsageType:=_UsedBySSW) then

              InitSSW := _SetTriggerUnits;
            end_if;
          else
            aProperties[0].udPropertyId     := SDM_PROP_TASK_CONTROL_DURATION_TIMEOUT;
            aProperties[0].udPropertyValue  := TaskConfig.TaskDurationTimeout_us;

            aProperties[1].udPropertyId     := SDM_PROP_TASK_CONTROL_CONFIGURATION;
            aProperties[1].udPropertyValue  := TaskConfig.Config;

            if SDIAS_iSetNodePropertiesIndex(hNodeHandle      := udNodeHandle
                                      , udIndex               := 2
                                      , udPropertyCount       := 2
                                      , psPropertyValuePairs  := #aProperties[0]
                                      ) = SDIAS_OK then

              InitSSW := _SetTriggerUnits;
            else
              LogError("(SdiasManager::CyWork) Failed to set the iso read start config via OS interface!");
              ErrorInitStep := InitSSW;
              InitSSW := _PrepareError;
              ClassState := _ManagerError;
            end_if;
          end_if;
        else
          LogError("(SdiasManager::CyWork) Couldn't find iso write entry in info block! Unable to continue with Initialisation!");
          ClassState := _ComponentNotExists;
          ErrorInitStep := InitSSW;
          InitSSW := _PrepareError;
        end_if;

//**********************************************************************************************************************************************************
      _SetTriggerUnits:
        // configure trigger unit 0 (use it for both iso tasks)
        TriggerUnitSetup[0].TaskSelect := 0;
        TriggerUnitSetup[0].TaskSelect.IsoWrite := TRUE;
        TriggerUnitSetup[0].TaskSelect.IsoRead  := FALSE; // for read task it's set later in realtime

        TriggerUnitSetup[0].StartAddress := ISOWriteDO.Offset; // trigger unit size has already been subtracted before
        TriggerUnitSetup[0].StartAddress.UnitEnable := TRUE;

        // configure trigger unit 1 for direct access
        TriggerUnitSetup[1].TaskSelect := 0;
        TriggerUnitSetup[1].TaskSelect.DirectAccess := TRUE;

        // search for the direct access read entry in the info block
        b_FoundIt := FALSE;
        for i := 0 to ManagerInfoBlock.MappingInfo.MappingInfoNo-1 do
          if ManagerInfoBlock.MappingInfo.aMappingInfos[i].MappingID = DAWrPayload then
            b_FoundIt := TRUE;
            exit;
          end_if;
        end_for;

        if b_FoundIt then
          TriggerUnitSetup[1].StartAddress := ManagerInfoBlock.MappingInfo.aMappingInfos[i].StartAddress;
          TriggerUnitSetup[1].StartAddress.UnitEnable := TRUE;

          WriteLength := sizeof(t_TriggerUnitSetupX2);
        else
          WriteLength := sizeof(t_TriggerUnitSetup);
          LogError("(SdiasManager::CyWork) Couldn't find the Direct Access Write Payload info in the module mapping");
        end_if;

        if ConnectionType = SDIAS_CON_VIA_VARAN_uC then

          // if the µC detects the setting on this address, it will stop to start the task in a loop (it starts again if the execution request
          ASYWriteDO.pData^$t_TriggerUnitSetupX2 := TriggerUnitSetup;
          if ChangeAsyWr(Offset:=SDIAS_OFFSET_TRIGGER_UNIT_SETUP_0,
                         Length:=WriteLength,
                         RunState:=_BUS_IF_RUN_STATE_SINGLE_RUN,
                         UsageType:=_UsedBySSW) then

#pragma warning(disable: 74)
            // for local SDIAS we set the enable bit for the watchdog trigger DO (must be enabled always)
            TempControlByte := 0;
            TempControlByte.EnableDO := TRUE;
#pragma warning(default: 74)
            (ISOWriteDO.pData$^t_SDIAS_ControlByte + SDIAS_TRIGGER_UNIT_BYTE_SIZE)^ := TempControlByte;

            b_WdTriggerActive := TRUE;
            ud_LastWdTime := ops.tAbsolute - SDIAS_WATCHDOG_TRIGGER_TIME - 1; // start with first watchdog now

            InitSSW := _WriteDAList;
          end_if;
        else
          aProperties[0].udPropertyId     := SDM_PROP_TASK_TRIGGER_UNIT_CONTROL;
          aProperties[0].udPropertyValue  := to_udint(TriggerUnitSetup[0].TaskSelect);

          aProperties[1].udPropertyId     := SDM_PROP_TASK_TRIGGER_UNIT_START_ADDR_RANGE;
          aProperties[1].udPropertyValue  := to_udint(TriggerUnitSetup[0].StartAddress);

          if SDIAS_iSetNodePropertiesIndex(hNodeHandle          := udNodeHandle
                                          , udIndex             := 0
                                          , udPropertyCount     := 2
                                          , psPropertyValuePairs:= #aProperties[0]
                                          ) = SDIAS_OK then

            aProperties[0].udPropertyId     := SDM_PROP_TASK_TRIGGER_UNIT_CONTROL;
            aProperties[0].udPropertyValue  := to_udint(TriggerUnitSetup[1].TaskSelect);

            aProperties[1].udPropertyId     := SDM_PROP_TASK_TRIGGER_UNIT_START_ADDR_RANGE;
            aProperties[1].udPropertyValue  := to_udint(TriggerUnitSetup[1].StartAddress);

            if SDIAS_iSetNodePropertiesIndex(hNodeHandle          := udNodeHandle
                                            , udIndex             := 1
                                            , udPropertyCount     := 2
                                            , psPropertyValuePairs:= #aProperties[0]
                                            ) = SDIAS_OK then

#pragma warning(disable: 74)
              // for local SDIAS we set the enable bit for the watchdog trigger DO (must be enabled always)
              TempControlByte := 0;
              TempControlByte.EnableDO := TRUE;
#pragma warning(default: 74)
              (ISOWriteDO.pData$^t_SDIAS_ControlByte + SDIAS_TRIGGER_UNIT_BYTE_SIZE)^ := TempControlByte;

              b_WdTriggerActive := TRUE;
              ud_LastWdTime := ops.tAbsolute - SDIAS_WATCHDOG_TRIGGER_TIME - 1; // start with first watchdog now

              InitSSW := _WriteDAList;
            else
              LogError("(SdiasManager::CyWork) Failed to make the trigger unit 2 settings via OS interface!");
              ErrorInitStep := InitSSW;
              InitSSW := _PrepareError;
              ClassState := _ManagerError;
            end_if;
          else
            LogError("(SdiasManager::CyWork) Failed to make the trigger unit 1 settings via OS interface!");
            ErrorInitStep := InitSSW;
            InitSSW := _PrepareError;
            ClassState := _ManagerError;
          end_if;
        end_if;

//**********************************************************************************************************************************************************
      _WriteDAList:
        // clear the list
        _memset(dest:=#DAListOfDOs, usByte:=0, cntr:=sizeof(DAListOfDOs));

        // initialize the module select array for module initialisation (maybe there are less modules to initialize than SDO channels available)
        NextPlace := 0;
        for i := 0 to SDIAS_SDO_CHANNEL_NO-1 do
          ActModule[i] := SDIAS_PLACE_NO_MODULE_ADDED_SO_FAR;
        end_for;

        // setup the command (memory access with 2 retries)
        DAListOfDOs[0].CmdRetries := 1 OR (2 SHL 5);

        // search for the da read payload entry in the info block
        b_FoundIt := FALSE;
        for i := 0 to ManagerInfoBlock.MappingInfo.MappingInfoNo-1 do
          if ManagerInfoBlock.MappingInfo.aMappingInfos[i].MappingID = DARdPayload then
            DAListOfDOs[0].OffsetReadPayload := ManagerInfoBlock.MappingInfo.aMappingInfos[i].StartAddress;
            b_FoundIt := TRUE;
            exit;
          end_if;
        end_for;

        if b_FoundIt = FALSE then
          LogError("(SdiasManager::CyWork) Couldn't find the Direct Access Read Payload info in the module mapping");
          InitSSW := _DeactivateSyncInjection;
          return;
        else
          b_FoundIt := FALSE;
        end_if;

        // search for the da write payload entry in the info block
        b_FoundIt := FALSE;
        for i := 0 to ManagerInfoBlock.MappingInfo.MappingInfoNo-1 do
          if ManagerInfoBlock.MappingInfo.aMappingInfos[i].MappingID = DAWrPayload then
            DAListOfDOs[0].OffsetWritePayload := ManagerInfoBlock.MappingInfo.aMappingInfos[i].StartAddress;
            b_FoundIt := TRUE;
            exit;
          end_if;
        end_for;

        if b_FoundIt = FALSE then
          LogError("(SdiasManager::CyWork) Couldn't find the Direct Access Write Payload info in the module mapping");
          InitSSW := _DeactivateSyncInjection;
          return;
        else
          b_FoundIt := FALSE;
        end_if;

        // search for the da list entry in the info block
        b_FoundIt := FALSE;
        for i := 0 to ManagerInfoBlock.MappingInfo.MappingInfoNo-1 do
          if ManagerInfoBlock.MappingInfo.aMappingInfos[i].MappingID = DAList then
            DAListOfDOs[0].OffsetWritePayload := ManagerInfoBlock.MappingInfo.aMappingInfos[i].StartAddress;
            b_FoundIt := TRUE;
            exit;
          end_if;
        end_for;

        if b_FoundIt = FALSE then
          LogError("(SdiasManager::CyWork) Couldn't find the Direct Access DO list info in the module mapping");
          InitSSW := _DeactivateSyncInjection;
          return;
        end_if;

        if ConnectionType = SDIAS_CON_VIA_VARAN_uC then
          // reset direct access read payload (toggle bits, error info)
          if ChangeAsyWr(Offset:=ManagerInfoBlock.MappingInfo.aMappingInfos[i].StartAddress,
                         Length:=128,
                         RunState:=_BUS_IF_RUN_STATE_SINGLE_RUN,
                         UsageType:=_UsedBySSW) then

            InitSSW := _ResetDARdPayload;
          end_if;
        else
          // OS already did this => skip the next step
          InitSSW := _ConfigDATask;
        end_if;

//**********************************************************************************************************************************************************
      _ResetDARdPayload:

        // reset the write buffer
        _memset(dest:=ASYWriteDO.pData, usByte:=0, cntr:=128);

        // search for the da read payload entry in the info block
        b_FoundIt := FALSE;
        for i := 0 to ManagerInfoBlock.MappingInfo.MappingInfoNo-1 do
          if ManagerInfoBlock.MappingInfo.aMappingInfos[i].MappingID = DARdPayload then
            DAListOfDOs[0].OffsetReadPayload := ManagerInfoBlock.MappingInfo.aMappingInfos[i].StartAddress;
            b_FoundIt := TRUE;
            exit;
          end_if;
        end_for;

        if b_FoundIt = FALSE then
          LogError("(SdiasManager::CyWork) Couldn't find the Direct Access Read Payload info in the module mapping");
          InitSSW := _DeactivateSyncInjection;
          return;
        end_if;

        // reset direct access read payload (toggle bits, error info)
        if ChangeAsyWr(Offset:=ManagerInfoBlock.MappingInfo.aMappingInfos[i].StartAddress,
                       Length:=128,
                       RunState:=_BUS_IF_RUN_STATE_SINGLE_RUN,
                       UsageType:=_UsedBySSW) then

          InitSSW := _ConfigDATask;
        end_if;

//**********************************************************************************************************************************************************
      _ConfigDATask:
        // search for the da list entry in the info block
        b_FoundIt := FALSE;
        for i := 0 to ManagerInfoBlock.MappingInfo.MappingInfoNo-1 do
          if ManagerInfoBlock.MappingInfo.aMappingInfos[i].MappingID = DAList then
            DAListOfDOs[0].OffsetWritePayload := ManagerInfoBlock.MappingInfo.aMappingInfos[i].StartAddress;
            b_FoundIt := TRUE;
            exit;
          end_if;
        end_for;

        // if we found it, use the offset in the task configuration
        if b_FoundIt then
          // initialize the write buffer for the direct access (the parts which stay the same)
          DaWriteBuffer.ContolByte := 0;
          DaWriteBuffer.ContolByte.EnableDO := TRUE;
          DaWriteBuffer.ContolByte.EnableFlexRead := TRUE;
          DaWriteBuffer.ContolByte.EnableFlexWrite := TRUE;

          // set the task duration limit
          TaskConfig.TaskDurationTimeout_us := (ud_BusTime_ns / 1000)$UINT;

          // start address of iso read list
          TaskConfig.Config := ManagerInfoBlock.MappingInfo.aMappingInfos[i].StartAddress;

          if ConnectionType = SDIAS_CON_VIA_VARAN_uC then

            ASYWriteDO.pData^$t_TaskConfig := TaskConfig;

            if ChangeAsyWr(Offset:=SDIAS_OFFSET_TASK_CONFIG_0,
                           Length:=sizeof(t_TaskConfig),
                           RunState:=_BUS_IF_RUN_STATE_SINGLE_RUN,
                           UsageType:=_UsedBySSW) then

              InitSSW := _DeactivateSyncInjection;
            end_if;
          else
            aProperties[0].udPropertyId     := SDM_PROP_TASK_CONTROL_DURATION_TIMEOUT;
            aProperties[0].udPropertyValue  := TaskConfig.TaskDurationTimeout_us;

            aProperties[1].udPropertyId     := SDM_PROP_TASK_CONTROL_CONFIGURATION;
            aProperties[1].udPropertyValue  := TaskConfig.Config;

            if SDIAS_iSetNodePropertiesIndex(hNodeHandle      := udNodeHandle
                                      , udIndex               := 0
                                      , udPropertyCount       := 2
                                      , psPropertyValuePairs  := #aProperties[0]
                                      ) = SDIAS_OK then
              InitSSW := _DeactivateSyncInjection;
            else
              LogError("(SdiasManager::CyWork) Failed to set the iso read start config via OS interface!");
              ErrorInitStep := InitSSW;
              InitSSW := _PrepareError;
              ClassState := _ManagerError;
            end_if;
          end_if;
        else
          LogError("(SdiasManager::CyWork) Couldn't find the Direct Access DO list info in the module mapping");

          InitSSW := _DeactivateSyncInjection;
        end_if;

//**********************************************************************************************************************************************************
      _DeactivateSyncInjection:
        // we select the read task for sync, there are no sync task trigger losses allowed and we leave the sync disabled
        SyncInjectionCfg := 16#02;

        if ConnectionType = SDIAS_CON_VIA_VARAN_uC then
          ASYWriteDO.pData^$t_SyncInjectionCfg := SyncInjectionCfg;

          if ChangeAsyWr(Offset:=SDIAS_OFFSET_SYNC_INJECTION_CFG,
                         Length:=sizeof(t_SyncInjectionCfg),
                         RunState:=_BUS_IF_RUN_STATE_SINGLE_RUN,
                         UsageType:=_UsedBySSW) then

            InitSSW := _PrepareModuleInitialisation;
          end_if;
        else
          aProperties[0].udPropertyId     := SDM_PROP_SYNC_INJECTION_CONFIG;
          aProperties[0].udPropertyValue  := SyncInjectionCfg;

          if SDIAS_iSetNodeProperties(hNodeHandle         := udNodeHandle
                                    , udPropertyCount     := 1
                                    , psPropertyValuePairs:= #aProperties[0]
                                    ) = SDIAS_OK then
            InitSSW := _PrepareModuleInitialisation;
          else
            LogError("(SdiasManager::CyWork) Failed to deactivate sync injection via OS interface!");
            ErrorInitStep := InitSSW;
            InitSSW := _PrepareError;
            ClassState := _ManagerError;
          end_if;
        end_if;

//**********************************************************************************************************************************************************
      _PrepareModuleInitialisation:
        // asy write DO can now be used for other purposes (will be used for module initialisation)
        AsyWriteUsage := _NotUsed;

        // wait for varan Manager to be ready, otherwise we can't get the module out of reset state
        if (ConnectionType = SDIAS_CON_VIA_VARAN_uC) & (b_PostInitFinished = FALSE) then
          // only if we're still in post init
          if b_PostInitFinished = FALSE then
            // tell the manager we're finished with DO creation
            tempCmd.uiCmd := _BUS_IF_DO_CREATION_FINISHED;
            ToBusInterface.NewInst(pPara:=#tempCmd, pResult:=#_result);
          end_if;

          if _result.aData[0]$t_BusIFRetvalErrorcode <> _BUS_IF_RETVAL_OK then
            LogError("(SdiasManager::CyWork) Failed to tell the manager that the DOs have been created");
          end_if;

          InitSSW := _Wait4OtherModules;
        else
          InitSSW := _Wait4HardwareReady;
        end_if;

//**********************************************************************************************************************************************************
      _Wait4OtherModules:
        // wait until all sdias managers have created their DOs => needed to create the Mov-DOs which copy safety SPDOs between the modules
        tempCmd.uiCmd := _BUS_IF_DO_MEM_READY;
        ToBusInterface.NewInst(pPara:=#tempCmd, pResult:=#_result);

        if _result.aData[0]$t_BusIFRetvalErrorcode <> _BUS_IF_RETVAL_OK then
          LogError("(SdiasManager::CyWork) Failed to tell the manager that the DOs have been created");
        else
          // if they are ready => continue
          if _result.aData[4] then

            // if the ISO DOs were created in this initialisation run => create move DOs
            if b_IsoDOsJustCreated then
              b_IsoDOsJustCreated := FALSE;

              // create move DOs
              tempCmd.uiCmd := SDIAS_CMD_DATA_POINTER_AVAILABLE;
              pModuleInfo := #ModuleObjInfo[0];
              for i := 0 to MaxPlace do
                // check only the available objects
                if pModuleInfo^.pThis then
                  if pModuleInfo^.pThis^.NewInst(pPara:=#tempCmd, pResult:=#_result) <> READY then
                    LogValue("(SdiasManager::CyWork) Initialisation of module at place 0x{0} failed! (Data pointers were available)", i);
                  end_if;
                end_if;

                pModuleInfo += sizeof(t_ModuleObjectInfo);
              end_for;
            end_if;

            // tell the manager we're finished with DO creation
            tempCmd.uiCmd := _BUS_IF_MOVE_DO_CREATION_FINISHED;
            ToBusInterface.NewInst(pPara:=#tempCmd, pResult:=#_result);

            InitSSW := _Wait4VaranManager;
          end_if;
        end_if;

//**********************************************************************************************************************************************************
      _Wait4VaranManager:
        // wait until all sdias managers have created their move DOs => needed to create the Mov-DOs which copy safety SPDOs between the modules
        tempCmd.uiCmd := _BUS_IF_MOVE_DO_MEM_READY;
        ToBusInterface.NewInst(pPara:=#tempCmd, pResult:=#_result);

        if _result.aData[0]$t_BusIFRetvalErrorcode <> _BUS_IF_RETVAL_OK then
          LogError("(SdiasManager::CyWork) Failed to tell the manager that the Move DOs have been created");
        else
          // if they are ready => continue
          if _result.aData[4] then
            InitSSW := _Wait4HardwareReady;
          end_if;
        end_if;

//**********************************************************************************************************************************************************
      _Wait4HardwareReady:
        // wait until init is finished and the modules are no longer in reset state (takes about 10ms, we wait 15ms)
        if DOStartTime & ((ops.tAbsolute - DOStartTime) >= SDIAS_HARDWARE_STARTUP_TIME) then

          // Find the first Module to initialize
          // Search before the loop over SDIAS_SDO_CHANNEL_NO, otherwise 1 channel will be unused.
          if ((ModuleObjInfo[NextPlace].pThis = NIL) | (ModuleObjInfo[NextPlace].pInitState^ <> _NotInitialized)) & MaxPlace then
            repeat
              // skip places, where we don't have to initialize something
              NextPlace += 1;
            until (ModuleObjInfo[NextPlace].pThis & (ModuleObjInfo[NextPlace].pInitState^ = _NotInitialized)) | (NextPlace = MaxPlace) end_repeat;
          end_if;

          // select the first x modules to initialize (x = number of available SDO channels)
          for i := 0 to SDIAS_SDO_CHANNEL_NO-1 do
            if ModuleObjInfo[NextPlace].pThis & (ModuleObjInfo[NextPlace].pInitState^ = _NotInitialized) then
              ActModule[i] := NextPlace;
              LastSelected := NextPlace;
              ModuleInitStartTime[i] := OS_READMICROSEC();
              if NextPlace < MaxPlace then
                repeat
                  // skip places, where we don't have to initialize something
                  NextPlace += 1;
                until (ModuleObjInfo[NextPlace].pThis & (ModuleObjInfo[NextPlace].pInitState^ = _NotInitialized)) | (NextPlace = MaxPlace) end_repeat;
              else
                exit;
              end_if;
            elsif (NextPlace < MaxPlace) then
              repeat
                // skip places, where we don't have to initialize something
                NextPlace += 1;
              until (ModuleObjInfo[NextPlace].pThis & (ModuleObjInfo[NextPlace].pInitState^ = _NotInitialized)) | (NextPlace = MaxPlace) end_repeat;
            end_if;
          end_for;

          // remember the last selected number to continue there in the next step
          NextPlace := LastSelected;

          InitSSW := _ModuleInitialisation;
        end_if;

//**********************************************************************************************************************************************************
      _ModuleInitialisation:
        // we can only initialize the modules if both asynchronous accesses are available
        if (AsyReadUsage = _NotUsed) & (AsyWriteUsage = _NotUsed) then

          // preinitialize the complete marker => is resetted if a module has to be initialized
          b_ModulInitComplete := TRUE;

          // post init blocks the tasks in cyclic priority (the SDIAS Manager Code is running in lower priority than cyclic and has no time during the postinit) => give it some time
          if (b_PostInitFinished = FALSE) then
            ToMultiTask.TASKDELAY(timeout0:=SDIAS_WAIT_TIME_IN_POST_INIT);
          end_if;

          // work parallel on all available channels
          for i := 0 to SDIAS_SDO_CHANNEL_NO-1 do
            b_ModulInitFinished := FALSE;
            // if we have selected a module at this position => initialize it
            if ActModule[i] <> SDIAS_PLACE_NO_MODULE_ADDED_SO_FAR then
              b_ModulInitComplete := FALSE;

              RetcodeIPR := ModuleObjInfo[ActModule[i]].pThis^.InitModule();

              if RetcodeIPR = ERROR then
                LogValue("(SdiasManager::CyWork) Failed to initialize module on SDIAS Place 0x{0} via InitModule-Interface", ActModule[i]);

                // if it's an required module => error
                if ModuleObjInfo[ActModule[i]].Required then
                  SetRequiredError(pTargetThis:=ModuleObjInfo[ActModule[i]].pThis, Place:=ActModule[i]);
                else
                  //otherwise continue with the next module
                  b_ModulInitFinished := TRUE;
                end_if;
              elsif RetcodeIPR = READY then
                b_ModulInitFinished := TRUE;
              end_if;

              if b_ModulInitFinished then
                // save duration for this module
                TempTime := OS_READMICROSEC();
                ModuleObjInfo[ActModule[i]].ModuleInitDuration_us := TempTime - ModuleInitStartTime[i];
                ModuleInitStartTime[i] := TempTime;

                if NextPlace < MaxPlace then
                  repeat
                    // skip places, where we don't have to initialize something
                    NextPlace += 1;
                  until (ModuleObjInfo[NextPlace].pThis & (ModuleObjInfo[NextPlace].pInitState^ = _NotInitialized)) | (NextPlace = MaxPlace) end_repeat;

                  // if we found something to initialize
                  if (ModuleObjInfo[NextPlace].pThis & (ModuleObjInfo[NextPlace].pInitState^ = _NotInitialized)) then
                    // remember it
                    ActModule[i] := NextPlace;
                  else
                    // otherwise we reached max place
                    ActModule[i] := SDIAS_PLACE_NO_MODULE_ADDED_SO_FAR;
                  end_if;
                else
                  // reached max place
                  ActModule[i] := SDIAS_PLACE_NO_MODULE_ADDED_SO_FAR;
                end_if;
              end_if;
            end_if;
          end_for;

          if b_ModulInitComplete then
            InitSSW := _SetActualLEDStates;
          end_if;
        end_if;

//**********************************************************************************************************************************************************
      _SetActualLEDStates:
        // asy write DO can now be used for other purposes (will be used for LEDs)
        AsyWriteUsage := _NotUsed;

        // write the LED States to the Hardware
        b_NewLEDStates := TRUE;

        InitSSW := _FinishInitialisation;

//**********************************************************************************************************************************************************
      _FinishInitialisation:
        // tell the manager that we're finished with initializing
        if b_PostInitFinished = FALSE then
          SendPostInitFinished();
        end_if;

        // now that we're finished, we take the Bitmap from the OS:
        // At plug in during runtime it will detect the connect-event later, therefore we take the new and the old value from OS => then we don't detect a disconnect because of this delay
        OldDeviceBitmap := HardwareConfig.DeviceBitmap;
        sd_retval := SDIAS_iGetBitmapOfDevices(uiMaster:=0, pucNode:=pHwPath, udBufferLength:=8, pucData:=(#HardwareConfig.DeviceBitmap)$^USINT);

        if sd_retval & (CyclicMsgMarker.AlreadyPosted.GetDeviceBitmap = FALSE) then
          LogValue("(SdiasManager::CyWork) SDIAS_iGetBitmapOfDevices failed with error code -0x{0}", ABS(sd_retval)$UDINT);
          CyclicMsgMarker.AlreadyPosted.GetDeviceBitmap := TRUE;
        end_if;

        InitDuration := ops.tAbsolute - InitStartTime;

        InitSSW := _WaitForRtOperational;

        // now we're ready to start the DOs
        RtSSW := _Wait4DOs;
        b_Ready4Rt := TRUE;

//**********************************************************************************************************************************************************
      _WaitForRtOperational:
        // wait to get finished by rt ssw

        // this step is to continue calling the cyclic for watchdog triggering but not call the single modules because that could lead to SDO timeouts

//**********************************************************************************************************************************************************
      _InitFinished:
        if MaxPlace <> SDIAS_PLACE_NO_MODULE_ADDED_SO_FAR then
          // refresh global SDIAS retry counter
          pModuleInfo := #ModuleObjInfo[0];
          for i := 0 to MaxPlace do
            if pModuleInfo^.pThis & (pModuleInfo^.pThis^.ClassState <> _NoHardware) & (pModuleInfo^.pThis^.ClassState <> _WrongHardware) then
              // update retrycounter
              if (pModuleInfo^.pThis^.RetryCounter > pModuleInfo^.OldRetryCounter) then
                RetryCounter += pModuleInfo^.pThis^.RetryCounter - pModuleInfo^.OldRetryCounter;
                pModuleInfo^.OldRetryCounter := pModuleInfo^.pThis^.RetryCounter;
              end_if;

              // call cywork of all objects which are marked for a cyclic call
              if pModuleInfo^.bCyclic then
                pModuleInfo^.pThis^.UpdateCy();
              end_if;
            end_if;
            pModuleInfo += sizeof(t_ModuleObjectInfo);
          end_for;

          // check for a change of the hardware configuration (should be plug and play)
          sd_retval := SDIAS_iGetBitmapOfDevices(uiMaster:=0, pucNode:=pHwPath, udBufferLength:=8, pucData:=(#HardwareConfig.DeviceBitmap)$^USINT);
          if sd_retval & (CyclicMsgMarker.AlreadyPosted.GetDeviceBitmap = FALSE) then
            LogValue("(SdiasManager::CyWork) SDIAS_iGetBitmapOfDevices failed with error code -0x{0}", ABS(sd_retval)$UDINT);
            CyclicMsgMarker.AlreadyPosted.GetDeviceBitmap := TRUE;
          end_if;

          if HardwareConfig.DeviceBitmap <> OldDeviceBitmap then
            // check for changes from 1 to 0 (module removed) and if the removed module is required
            CompareBitmap[0] := HardwareConfig.DeviceBitmap[0] XOR 16#FFFFFFFF; // we want only the 0s in the new bitmap
            CompareBitmap[1] := HardwareConfig.DeviceBitmap[1] XOR 16#FFFFFFFF; // we want only the 0s in the new bitmap

            ResultBitmap[0] := OldDeviceBitmap[0] AND CompareBitmap[0]; // now we check for the 1=>0 switch
            ResultBitmap[1] := OldDeviceBitmap[1] AND CompareBitmap[1]; // now we check for the 1=>0 switch

            // if a module has been plugged off
            if ResultBitmap[0] | ResultBitmap[1] then

              pModuleInfo := #ModuleObjInfo[0];
              for i := 0 to MaxPlace do
                // check only the available objects
                if pModuleInfo^.pThis then
                  if i < 32 then
                    // in first 32 places
                    if ResultBitmap[0] AND (1 SHL i) then
                      pModuleInfo^.pThis^.DisconnectEvent();
                      if pModuleInfo^.Required then
                        SetRequiredError(pTargetThis:=pModuleInfo^.pThis, Place:=i);
                      else
                        pModuleInfo^.pThis^.ClassState := _NoHardware;
                      end_if;
                    end_if;
                  else
                    // in last 32 places
                    if ResultBitmap[1] AND (1 SHL (i-32)) then
                      pModuleInfo^.pThis^.DisconnectEvent();
                      if pModuleInfo^.Required then
                        SetRequiredError(pTargetThis:=pModuleInfo^.pThis, Place:=i);
                      else
                        pModuleInfo^.pThis^.ClassState := _NoHardware;
                      end_if;
                    end_if;
                  end_if;
                end_if;

                pModuleInfo += sizeof(t_ModuleObjectInfo);
              end_for;
            end_if;

            OldDeviceBitmap := HardwareConfig.DeviceBitmap;
          end_if;
        end_if;

//**********************************************************************************************************************************************************
//**                ERROR HANDLING                                           *******************************************************************************
//**********************************************************************************************************************************************************
      _PrepareError: // do error handling and then stay in _ErrorOccured-Step
        // no watchdog triggering in error case
        b_WdTriggerActive := FALSE;
        ToggleReadTaskActive := FALSE;

        if b_MultipleConnectInInit then
          LogError("(SdiasManager::CyWork) Connect has been called twice during initialisation!");
        end_if;

        // tell the manager that we're finished with initializing
        if b_PostInitFinished = FALSE then
          SendPostInitFinished(DisableThisObject:=TRUE);
        end_if;

        // set required error, if there is a required module
        SetRequiredError();
(*
        // if no required error => set error according to class state
        tempCmd.uiCmd := _BUS_IF_SET_ERROR;
        tempCmd.aPara[0] := ClassState$DINT;

#ifdef HWK_SHOW_PRAGMA_MESSAGES
#pragma message("RamAnd 03.12.2013 18:15 \ Je nach Fehler die entsprechende Meldung ausgeben. tempCmd.aPara[1] soll den Pointer auf den String beinhalten")
#pragma message("RamAnd 03.12.2013 18:15 \ Wenn via VARAN Verbunden noch <exec climsg 45 > an den String vorne hinzufügen")
#pragma message("RamAnd 09.12.2013 17:14 \ Unterscheiden, ob abgestürzt werden soll (je nach Fehler und Required-Einstellung)")
#endif

        tempCmd.aPara[1] := 0;

        // only set an error if there are modules projected
        if (ClassState <> _NoHardware) & (MaxPlace <> SDIAS_PLACE_NO_MODULE_ADDED_SO_FAR) then
          ToBusInterface.NewInst(pPara:=#tempCmd, pResult:=#_result);
        end_if;

        if _result.aData[0]$t_BusIFRetvalErrorcode <> _BUS_IF_RETVAL_OK then
          LogError("(SdiasManager::CyWork) Failed to set an error to the bus interface!");
        end_if;
*)
        // if it's still running => stop the asy DOs
        ChangeAsyWr(Offset:=0,
                    Length:=0,
                    RunState:=_BUS_IF_RUN_STATE_NO_RUN,
                    UsageType:=AsyWriteUsage);

        ChangeAsyRd(Offset:=0,
                    Length:=0,
                    RunState:=_BUS_IF_RUN_STATE_NO_RUN,
                    UsageType:=AsyReadUsage);

        InitSSW := _ErrorOccured;

//**********************************************************************************************************************************************************
      _ErrorOccured: // do nothing here
        return;
//**********************************************************************************************************************************************************
    end_case;

    // SDO Handling (has to be done also during initialisation)
    CyclicSDOHandling();

    // we have to do this after SDO Handling, so we don't block the channel for SDOs with LED Infos
    if InitSSW = _InitFinished then
      // Appli LED State Handling
      if (AsyWriteUsage = _NotUsed) & (b_SendWdTrigger = FALSE) then
        // check if the LED Status has changed on any Module
        if b_NewLEDStates then
          if ConnectionType = SDIAS_CON_VIA_VARAN_uC then
            // write the new LED States to the Hardware
            ASYWriteDO.pData^$t_AppliLEDStates := AppliLEDStates;
            if ChangeAsyWr(Offset:=SDIAS_OFFSET_APPLI_LED_STATES,
                           Length:=sizeof(t_AppliLEDStates),
                           RunState:=_BUS_IF_RUN_STATE_SINGLE_RUN,
                           UsageType:=_UsedByLED) = FALSE then
              LogError("(SdiasManager::CyWork) Error occured at setting new Appli LED states");
            end_if;
          else
            aProperties[0].udPropertyId     := SDM_PROP_BITMAP_APPLICATION_LED_0_15;
            aProperties[0].udPropertyValue  := AppliLEDStates[0]$UDINT;

            aProperties[1].udPropertyId     := SDM_PROP_BITMAP_APPLICATION_LED_16_31;
            aProperties[1].udPropertyValue  := AppliLEDStates[4]$UDINT;

            aProperties[2].udPropertyId     := SDM_PROP_BITMAP_APPLICATION_LED_32_47;
            aProperties[2].udPropertyValue  := AppliLEDStates[8]$UDINT;

            aProperties[3].udPropertyId     := SDM_PROP_BITMAP_APPLICATION_LED_48_63;
            aProperties[3].udPropertyValue  := AppliLEDStates[12]$UDINT;

            if SDIAS_iSetNodeProperties(hNodeHandle         := udNodeHandle
                                      , udPropertyCount     := 4
                                      , psPropertyValuePairs:= #aProperties[0]
                                      ) <> SDIAS_OK then
              LogError("(SdiasManager::CyWork) Failed to set the application LED states via OS interface!");
              ErrorInitStep := InitSSW;
              InitSSW := _PrepareError;
              ClassState := _ManagerError;
            else
              b_NewLEDStates := FALSE;
            end_if;
          end_if;
        end_if;
      elsif AsyWriteUsage = _UsedByLED then
        b_NewLEDStates := FALSE;
        AsyWriteUsage := _NotUsed;
      end_if;
    elsif (b_PostInitFinished = FALSE) & InitStartTime & ((ops.tAbsolute - InitStartTime) > (SDIAS_INIT_BLOCK_TIMEOUT + AdditionalPostInitTime)) then
      // timeout for last init if we're stuck in a step for too long (1min). otherwise the plc would not start up, which makes it hard to show the error
      LogValue("(SdiasManager::CyWork) Init has been blocked for too long! Initialisation of SDIAS Manager timed out! Blocked step: 0x{0}",InitSSW$UDINT);
      ClassState := _TimeoutInInit;
      ErrorInitStep := InitSSW;
      InitSSW := _PrepareError;
    end_if;

  elsif b_PostInitFinished = FALSE then
    // if the module is not online => tell the manager that we're finished with initializing
    SendPostInitFinished(DisableThisObject:=TRUE);

    // set required error, if there is a required module
    SetRequiredError();
  end_if;

  PostRtMessages();

	state := READY;

END_FUNCTION

FUNCTION VIRTUAL GLOBAL SdiasManager::RtWork
	VAR_INPUT
		EAX 	: UDINT;
	END_VAR
	VAR_OUTPUT
		state (EAX) 	: UDINT;
	END_VAR
  VAR
  	calloption          : UDINT;
    i                   : UDINT;
    pModuleInfo         : ^t_ModuleObjectInfo;
    dataSETRUNSTATE     : t_SetRunStateCfg;
    dataSyncData        : t_SyncData;
  	tempCmd             : CmdStruct;
    _result             : results;
    pHelpAccess         : ^t_AccessElement;
    CheckRetryCounters  : BOOL;
    ActFrameCounter     : UDINT;
    TempControlByte     : t_SDIAS_ControlByte;
    dataUPDATEDO        : t_UpdateDOCfg;
    aProperties         : ARRAY [0..4] OF SDM_PROPERTY_VALUE_PAIR;
    SyncInjectionCfg    : t_SyncInjectionCfg;
    CrashThisTime       : USINT;
    aCrashMessage       : ARRAY [0..255] OF CHAR;
    TmpRetryCount       : UDINT;
#ifdef SDIAS_RT_TIME_MEASUREMENT
    Time1           : UDINT;
    Time2           : UDINT;
    TimeTotal1      : UDINT;
    TimeTotal2      : UDINT;
#endif
  END_VAR

  // Called from BusInterface on UpdateRt or UpdateRtPostScan

  // Save state
  // This must be the 1. line in this function or EAX may be overwriten by the generated AWL code
  calloption := EAX;

  if Online then
    pModuleInfo := #ModuleObjInfo[0];
    case RtSSW of
//**********************************************************************************************************************************************************
      _RtIdle: // nothing

//**********************************************************************************************************************************************************
      _CreateAndModifyDOs: // create and modify ISO DOs
        CreateAndModifyIsoDOs();

        RtSSW := _Wait4DOs;

//**********************************************************************************************************************************************************
      _Wait4DOs:
        if calloption = CALL_OPTION_RT_PRESCAN then    // Called from UpdateRt
          // wait until the DOs can be activated
          if b_Ready4Rt then
            // activate the ISO DOs

            // general settings needed for all DOs
            dataSETRUNSTATE.NewRunState := _BUS_IF_RUN_STATE_CONT_RUN;
            tempCmd.uiCmd         := _BUS_IF_SET_RUN_STATE;
            tempCmd.aPara[0]      := (#dataSETRUNSTATE)$DINT;

#ifndef SDIAS_DEACTIVATE_TASK_CHECKS
            if ConnectionType = SDIAS_CON_VIA_VARAN_uC then
              // set runstate of taskinfo read
              dataSETRUNSTATE.Handle      := TaskInfoDO.Handle;

              ToBusInterface.NewInst(pPara:=#tempCmd, pResult:=#_result);

              if _result.aData[0]$t_BusIFRetvalErrorcode <> _BUS_IF_RETVAL_OK then
                // remember the log message and write it in cyclic priority to avoid a rt runtime error
                CyclicMsgMarker.PostIt.TaskInfoRunFailed := TRUE;
              end_if;
            end_if;
#endif

            // set runstate of read
            dataSETRUNSTATE.Handle      := ISOReadDO.Handle;

            ToBusInterface.NewInst(pPara:=#tempCmd, pResult:=#_result);

            if _result.aData[0]$t_BusIFRetvalErrorcode <> _BUS_IF_RETVAL_OK then
              // remember the log message and write it in cyclic priority to avoid a rt runtime error
              CyclicMsgMarker.PostIt.IsoReadRunFailed := TRUE;
            end_if;

            // set runstate of write
            dataSETRUNSTATE.Handle      := ISOWriteDO.Handle;

            ToBusInterface.NewInst(pPara:=#tempCmd, pResult:=#_result);

            if _result.aData[0]$t_BusIFRetvalErrorcode <> _BUS_IF_RETVAL_OK then
              // remember the log message and write it in cyclic priority to avoid a rt runtime error
              CyclicMsgMarker.PostIt.IsoWriteRunFailed := TRUE;
            end_if;

            if ConnectionType = SDIAS_CON_VIA_VARAN_uC then

              // change config DO => change task config settings for Iso Read Task)
              ISOConfigWrDO.Offset := SDIAS_OFFSET_TASK_CONFIG_1;
              ISOConfigWrDO.Length := sizeof(t_TaskConfig);

              dataUPDATEDO.Handle               := ISOConfigWrDO.Handle;
              dataUPDATEDO.ud_addressoff_write  := ISOConfigWrDO.Offset;
              dataUPDATEDO.ud_length_write      := ISOConfigWrDO.Length;

              tempCmd.uiCmd         := _BUS_IF_UPDATE_DO;
              tempCmd.aPara[0]      := (#dataUPDATEDO)$DINT;

              ToBusInterface.NewInst(pPara:=#tempCmd, pResult:=#_result);

              if _result.aData[0]$t_BusIFRetvalErrorcode <> _BUS_IF_RETVAL_OK then
                // remember the log message and write it in cyclic priority to avoid a rt runtime error
                CyclicMsgMarker.PostIt.IsoConfigWrChangeFailed := TRUE;
              else
                // use the task config data
                ISOConfigWrDO.pData^$t_TaskConfig := ISOTaskConfig;
              end_if;

              dataSETRUNSTATE.NewRunState := _BUS_IF_RUN_STATE_SINGLE_RUN;
              dataSETRUNSTATE.Handle      := ISOConfigWrDO.Handle;

              tempCmd.uiCmd               := _BUS_IF_SET_RUN_STATE;
              tempCmd.aPara[0]            := (#dataSETRUNSTATE)$DINT;

              ToBusInterface.NewInst(pPara:=#tempCmd, pResult:=#_result);

              if _result.aData[0]$t_BusIFRetvalErrorcode <> _BUS_IF_RETVAL_OK then
                // remember the log message and write it in cyclic priority to avoid a rt runtime error
                CyclicMsgMarker.PostIt.IsoConfigWrTaskConfigFailed := TRUE;
              end_if;

            else
              aProperties[0].udPropertyId     := SDM_PROP_TASK_CONTROL_DURATION_TIMEOUT;
              aProperties[0].udPropertyValue  := ISOTaskConfig.TaskDurationTimeout_us;

              aProperties[1].udPropertyId     := SDM_PROP_TASK_CONTROL_CONFIGURATION;
              aProperties[1].udPropertyValue  := ISOTaskConfig.Config;

              if SDIAS_iSetNodePropertiesIndex(hNodeHandle      := udNodeHandle
                                        , udIndex               := 1
                                        , udPropertyCount       := 2
                                        , psPropertyValuePairs  := #aProperties[0]
                                        ) <> SDIAS_OK then
                CyclicMsgMarker.PostIt.IsoTaskConfigFailed := TRUE;
              end_if;

              // reconfigure PLL to ensure the SDIAS Sync refers to the correct OS tick

              // get the actual frame counter
              if SDIAS_iGetNodeProperty(hNodeHandle      :=udNodeHandle
                                      , udPropertyId     :=SDM_PROP_PLL_SYNC_TIME_FRAME_COUNTER
                                      , pudPropertyValue :=#ActFrameCounter
                                      ) = SDIAS_OK then

                tempCmd.uiCmd := _BUS_IF_SET_SYNC;

                dataSyncData.us_sync_nr := SDIAS_EVENT_MASK_ID_SYNC_OUT2; // iso read trigger
                dataSyncData.us_period_multiplier := 0;
                dataSyncData.sd_offset := 0;

                // start with the next correct sync
                dataSyncData.us_frame_count_threshold := (ActFrameCounter + 1 + (ud_BusTime_ns / 1000) / ud_SystemPeriodTime)$USINT;
                dataSyncData.us_enable_frame_count := 1;

                tempCmd.aPara[0] := (#dataSyncData)$DINT;

                ToBusInterface.NewInst(pPara:=#tempCmd, pResult:=#_result);

                if _result.aData[0]$t_BusIFRetvalErrorcode <> _BUS_IF_RETVAL_OK then
                  CyclicMsgMarker.PostIt.SetSyncFailed := TRUE;
                end_if;
              else
                CyclicMsgMarker.PostIt.GetFrameCounterFailed := TRUE;
              end_if;
            end_if;

            // stop asynchron watchdog triggering, because the watchdog gets triggered by rt now
            b_WdTriggerActive := FALSE;
            ToggleReadTaskActive := FALSE;
            b_SendWdTrigger := FALSE;

            if AsyWriteUsage = _UsedByWD then
              AsyWriteUsage := _NotUsed;
            end_if;

            PreOpCount := 0;
            RtSSW := _Wait4PllSync;
          end_if;
        end_if;

//**********************************************************************************************************************************************************
      _Wait4PllSync:
        if calloption = CALL_OPTION_RT_PRESCAN then    // Called from UpdateRt
          if PreOpCount < SDIAS_CYCLES_WAIT_AFTER_SYNC_ENABLE-1 then
            PreOpCount += 1;
          else
            PreOpCount := 0;
            RtSSW := _Wait2Ticks;
          end_if;
        end_if;

//**********************************************************************************************************************************************************
      _Wait2Ticks:  // SDIAS Manager FPGA measures the sync interval during the first to cycles
        if calloption = CALL_OPTION_RT_PRESCAN then    // Called from UpdateRt
          if PreOpCount < (SDIAS_SYNC_MEASURE_TICKS-1) then
            PreOpCount += 1;

            // we select the read task for sync, there are no sync task trigger losses allowed and we enable the sync injection
            SyncInjectionCfg := 16#03;

            if ConnectionType = SDIAS_CON_VIA_VARAN_uC then
              // change config DO => change trigger unit settings (also use trigger unit for read task)
              ISOConfigWrDO.Offset := SDIAS_OFFSET_SYNC_INJECTION_CFG;
              ISOConfigWrDO.Length := sizeof(t_SyncInjectionCfg);

              dataUPDATEDO.Handle               := ISOConfigWrDO.Handle;
              dataUPDATEDO.ud_addressoff_write  := ISOConfigWrDO.Offset;
              dataUPDATEDO.ud_length_write      := ISOConfigWrDO.Length;

              tempCmd.uiCmd         := _BUS_IF_UPDATE_DO;
              tempCmd.aPara[0]      := (#dataUPDATEDO)$DINT;

              ToBusInterface.NewInst(pPara:=#tempCmd, pResult:=#_result);

              if _result.aData[0]$t_BusIFRetvalErrorcode <> _BUS_IF_RETVAL_OK then
                // remember the log message and write it in cyclic priority to avoid a rt runtime error
                CyclicMsgMarker.PostIt.IsoConfigWrChange2Failed := TRUE;
              else
                // use the sync injection data
                ISOConfigWrDO.pData^$t_SyncInjectionCfg := SyncInjectionCfg;
              end_if;

              dataSETRUNSTATE.NewRunState := _BUS_IF_RUN_STATE_SINGLE_RUN;
              tempCmd.uiCmd               := _BUS_IF_SET_RUN_STATE;
              tempCmd.aPara[0]            := (#dataSETRUNSTATE)$DINT;

              dataSETRUNSTATE.Handle      := ISOConfigWrDO.Handle;

              ToBusInterface.NewInst(pPara:=#tempCmd, pResult:=#_result);

              if _result.aData[0]$t_BusIFRetvalErrorcode <> _BUS_IF_RETVAL_OK then
                // remember the log message and write it in cyclic priority to avoid a rt runtime error
                CyclicMsgMarker.PostIt.IsoConfigWrSyncInjFailed := TRUE;
              end_if;
            else
              aProperties[0].udPropertyId     := SDM_PROP_SYNC_INJECTION_CONFIG;
              aProperties[0].udPropertyValue  := SyncInjectionCfg;

              if SDIAS_iSetNodeProperties(hNodeHandle         := udNodeHandle
                                        , udPropertyCount     := 1
                                        , psPropertyValuePairs:= #aProperties[0]
                                        ) <> SDIAS_OK then
                // remember the log message and write it in cyclic priority to avoid a rt runtime error
                CyclicMsgMarker.PostIt.IsoSyncInjFailed := TRUE;
              end_if;
            end_if;
          else
            if ConnectionType = SDIAS_CON_VIA_VARAN_uC then
              // change config DO => change trigger unit settings (also use trigger unit for read task)
              ISOConfigWrDO.Offset := SDIAS_OFFSET_TRIGGER_UNIT_SETUP_0;
              ISOConfigWrDO.Length := sizeof(t_TriggerUnitSetup);

              dataUPDATEDO.Handle               := ISOConfigWrDO.Handle;
              dataUPDATEDO.ud_addressoff_write  := ISOConfigWrDO.Offset;
              dataUPDATEDO.ud_length_write      := ISOConfigWrDO.Length;

              tempCmd.uiCmd         := _BUS_IF_UPDATE_DO;
              tempCmd.aPara[0]      := (#dataUPDATEDO)$DINT;

              ToBusInterface.NewInst(pPara:=#tempCmd, pResult:=#_result);

              if _result.aData[0]$t_BusIFRetvalErrorcode <> _BUS_IF_RETVAL_OK then
                // remember the log message and write it in cyclic priority to avoid a rt runtime error
                CyclicMsgMarker.PostIt.IsoConfigWrChangeFailed := TRUE;
              else
                // use the trigger unit setup data
                ISOConfigWrDO.pData^$t_TriggerUnitSetup := ISOTriggerUnitSetup;
              end_if;

              dataSETRUNSTATE.NewRunState := _BUS_IF_RUN_STATE_SINGLE_RUN;
              tempCmd.uiCmd               := _BUS_IF_SET_RUN_STATE;
              tempCmd.aPara[0]            := (#dataSETRUNSTATE)$DINT;

              dataSETRUNSTATE.Handle      := ISOConfigWrDO.Handle;

              ToBusInterface.NewInst(pPara:=#tempCmd, pResult:=#_result);

              if _result.aData[0]$t_BusIFRetvalErrorcode <> _BUS_IF_RETVAL_OK then
                // remember the log message and write it in cyclic priority to avoid a rt runtime error
                CyclicMsgMarker.PostIt.IsoConfigWrTriggerUnitFailed := TRUE;
              end_if;
            else
              aProperties[0].udPropertyId     := SDM_PROP_TASK_TRIGGER_UNIT_CONTROL;
              aProperties[0].udPropertyValue  := to_udint(ISOTriggerUnitSetup.TaskSelect);

              aProperties[1].udPropertyId     := SDM_PROP_TASK_TRIGGER_UNIT_START_ADDR_RANGE;
              aProperties[1].udPropertyValue  := to_udint(ISOTriggerUnitSetup.StartAddress);

              if SDIAS_iSetNodePropertiesIndex(hNodeHandle          := udNodeHandle
                                              , udIndex             := 0
                                              , udPropertyCount     := 2
                                              , psPropertyValuePairs:= #aProperties[0]
                                              ) <> SDIAS_OK then
                CyclicMsgMarker.PostIt.IsoTriggerUnitConfigFailed := TRUE;
              end_if;
            end_if;

            // tell the manager that our sync is running, which triggers the watchdog on the modules from now on
            tempCmd.uiCmd := _BUS_IF_RT_SYNC_READY;
            ToBusInterface.NewInst(pPara:=#tempCmd, pResult:=#_result);

            // sync is starting with this RT => deactivate the watchdog trigger (no longer needed)
  #pragma warning(disable: 74)
            TempControlByte := 0;
            TempControlByte.EnableDO := FALSE;
  #pragma warning(default: 74)
            (ISOWriteDO.pData$^t_SDIAS_ControlByte + SDIAS_TRIGGER_UNIT_BYTE_SIZE)^ := TempControlByte;

            PreOpCount := 0;
            RtSSW := _PreOperational;
          end_if;
        end_if;

//**********************************************************************************************************************************************************
      _PreOperational: // we have to make 1 step between start of DOs and operational => task status bits are not valid the first time
        if calloption = CALL_OPTION_RT_PRESCAN then    // Called from UpdateRt
          if PreOpCount < SDIAS_TASKINFO_READY_TICKS then
            PreOpCount += 1;
          else
            // finalize cyclic ssw
            if InitSSW = _WaitForRtOperational then
              ClassState  := _ClassOk;
              InitSSW     := _InitFinished;
              if ConnectionType = SDIAS_CON_VIA_VARAN_uC then
                // data is valid -> set online server to 1
                tempCmd.uiCmd    := _BUS_IF_SET_ONLINE;
                tempCmd.aPara[0] := 1;

                ToBusInterface.NewInst(pPara:=#tempCmd, pResult:=#_result);

                if _result.aData[0]$t_BusIFRetvalErrorcode <> _BUS_IF_RETVAL_OK then
                  // remember the log message and write it in cyclic priority to avoid a rt runtime error
                  CyclicMsgMarker.PostIt.SetOnlineStateFailed := TRUE;
                end_if;
              end_if;
            end_if;

            RtSSW := _Operational;

            //Set Classstates of the single modules and call the UpdateRt method to ensure valid data on the module servers if we set the state to _ClassOk.
            for i := 0 to MaxPlace do
              if pModuleInfo^.pThis then
                if pModuleInfo^.pInitState then

                  //Set ClassState of module, before calls of UpdateRt, since there are some modules which check the classstate in the UpdateRt Method
                  pModuleInfo^.pThis^.ClassState := pModuleInfo^.pInitState^;

                  if pModuleInfo^.bPreScan & (pModuleInfo^.pInitState^ = _ClassOk) then
                    // call all objects which are marked for prescan, to ensure valid data on user if classtate is class ok
                    pModuleInfo^.pThis^.UpdateRt();
                  end_if;
                else
                 //not possible
                end_if;
              end_if;
              pModuleInfo += sizeof(t_ModuleObjectInfo);
            end_for;
          end_if;
